FUNCTION_BLOCK T_RoboConnect_SetDigitalOutput_IncorrectIndexFails EXTENDS T_UnitTestBase
VAR
  robot : I_RoboConnect;
  targetDO : UINT;
  myTestState, prevState :
    (INIT, ARRANGE, ACT, ASSERT) := INIT;
  expected : BOOL;
  actual : BOOL := TRUE;
  counter : UINT;
END_VAR

CASE myTestState OF
  INIT:
    StateChanged();
    myTestState := ARRANGE;

  ARRANGE:
    IF StateChanged() THEN
      expected := FALSE;
      myTestState := ACT;
    END_IF

  ACT:
    actual := robot.SetDigitalOutput(targetDO, TRUE);
    myTestState := ASSERT;

  ASSERT:
    actual := robot.GetDigitalOutput(targetDO);
    assertion.AssertEquals_BOOL(expected, actual, 'actual := robot.SetDigitalOutput(targetDO, TRUE)');
    TestFinished();
    myTestState := INIT;

END_CASE

METHOD FB_init : BOOL
VAR_INPUT
  bInitRetains : BOOL; // if TRUE, the retain variables are initialized (warm start / cold start)
  bInCopyCode : BOOL; // if TRUE, the instance afterwards gets moved into the copy code (online change)
  TestSuite : tcl_SimpleUnitTestLibrary.I_TestSuite;
  robot : I_TcRobot;
  targetDo : UINT;
END_VAR
THIS^.robot := robot;
THIS^.targetDo := targetDo;
END_METHOD

METHOD PRIVATE StateChanged : BOOL
IF  myTestState = prevState THEN
  RETURN;
END_IF

prevState := myTestState;
StateChanged := TRUE;
END_METHOD

METHOD WaitForCycles : BOOL
VAR_INPUT
  maxCount : UINT;
END_VAR
counter := counter + 1;

IF counter = maxCount THEN
  counter := 0;
  WaitForCycles := TRUE;
END_IF
END_METHOD

END_FUNCTION_BLOCK

(* stored: Version 1.1.0.1
   POU T_TcRobot_SetDigitalOutput_IncorrectIndexFails: Id {78e09e6e-3b74-42a3-b419-0a9ef140c887}, SpecialFunc None
   Method FB_init: Id {9a516327-3b79-4929-8f53-9a02f0946c6c}
   Method StateChanged: Id {d7e52b9b-6c12-403f-8d22-2ecfd3cd7110}
   Method WaitForCycles: Id {721cecad-baa9-4653-b7e7-fa362ff3d34b} *)
